FUNCTION_BLOCK FB_Pushover
VAR_INPUT
    bSend                : BOOL;
    sToken               : STRING(30);
	sUser				 : STRING(30);
	sMessage			 : STRING(180);
	sDevice				 : STRING(20);
	sTitle				 : STRING(20);
	iPriority			 : DINT;
END_VAR
VAR_IN_OUT
    fbClient             : FB_IotHttpClient;
END_VAR
VAR_OUTPUT
    bBusy                : BOOL;
    bError               : BOOL;
END_VAR
VAR
    fbRequest            : FB_IotHttpRequest;
    fbJson               : FB_JsonDomParser;
    fbJsonWriter         : FB_JsonSaxWriter;
    nState               : UDINT;
    RisingEdge           : R_TRIG;
    
    bGetContentResult    : BOOL;
    sContent             : STRING(511);
    sSend                : STRING(511);
    
    bGetJsonResult       : BOOL;
    jsonDoc              : SJsonValue;
    jsonVal              : SJsonValue;
    sResultValue         : STRING;
    
    nReqCount            : UDINT;    
    nResCount            : UDINT;
    nValidResCount       : UDINT;
    nErrCount            : UDINT;
    
    fbTimer              : TON;
    bLightOn             : BOOL;
	iResponseStatus		 : DINT;
END_VAR

RisingEdge(CLK:= bSend );
CASE nState OF
0:    
        fbJsonWriter.StartObject();
		fbJsonWriter.AddKeyString('token',sToken );
        fbJsonWriter.AddKeyString('user',sUser);
		IF LEN(sTitle) <> 0 THEN
		fbJsonWriter.AddKeyString('title', sTitle);
		END_IF
		IF LEN(sDevice) <> 0 THEN
		fbJsonWriter.AddKeyString('device', sDevice);	
		END_IF
		fbJsonWriter.AddKeyNumber('priority', iPriority);
        fbJsonWriter.AddKeyString('message', sMessage);
        fbJsonWriter.EndObject();
        sSend:=fbJsonWriter.GetDocument();
        fbJsonWriter.ResetDocument();	
		fbRequest.sContentType := 'application/json';

    IF RisingEdge.Q THEN 

		IF fbRequest.SendRequest(sUri:='https://api.pushover.net/1/messages.json', fbClient:=fbClient, eRequestType:=ETcIotHttpRequestType.HTTP_POST, 
            pContent:=ADR(sSend), nContentSize:=LEN2(ADR(sSend)), 0) THEN                
            nState:= 1;
            nReqCount:= nReqCount+1;
            bBusy:= TRUE;
            bError:= FALSE;
        END_IF  
	END_IF
1:
    IF NOT fbRequest.bBusy THEN
        bError:= TRUE;
        IF NOT fbRequest.bError THEN                 
            bGetContentResult:= fbRequest.GetContent(pContent:= ADR(sContent), nContentSize:= SIZEOF(sContent), bSetNullTermination:= TRUE);
            IF fbRequest.nStatusCode >= 200 AND fbRequest.nStatusCode < 300 THEN
                bGetJsonResult:= FALSE;
                jsonDoc:= fbRequest.GetJsonDomContent(fbJson);
                IF jsonDoc <> 0 THEN
                    IF fbJson.HasMember(jsonDoc, 'status') THEN
                        jsonVal:= fbJson.FindMember(jsonDoc, 'status');
                        iResponseStatus := fbJson.GetInt(jsonVal);
                        IF iResponseStatus = 1 THEN
                            nValidResCount:= nValidResCount+1;
                            bError:= FALSE;
                        END_IF
                    END_IF		

					; // do something with status response
                    //nValidResCount:= nValidResCount+1;
                    //bError:= FALSE;    
                END_IF                            
                nResCount:= nResCount+1;            
            END_IF
        END_IF
        nState:= 0;
        bBusy:= FALSE;
        IF bError THEN
            nErrCount:= nErrCount+1;
        END_IF
    END_IF      
END_CASE

END_FUNCTION_BLOCK

(* stored: Version 1.1.0.1, ProductVersion 3.1.4024.13
   POU FB_Pushover: Id {31b5f6f1-ac80-462a-b777-5133763b4c37}, SpecialFunc None *)
